ABB RobotStudio station: Proy_ROBG.rspag

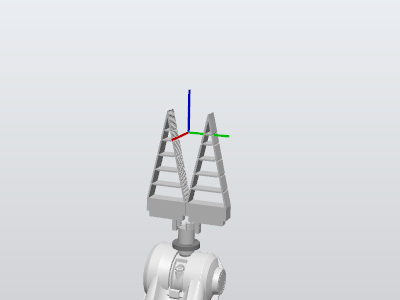
--- station ---
Station Project1 (saved by RobotStudio 23.3.10550.0)
Controller IRB140_6_81
  mechanical unit ROB_1: IRB140_6_81_C_03, 6 joints, base frame (0, 0, 0) mm
Layout (positions relative to the parent item):
  - IRB140_6_81_C_03 [mechanism, from %ABB.RobotStudio.Models.IRB140%\IRB140_6_81_C_G_03.rslib] at (0, 0, 0) mm; joint values [0, 0, -2.1624, 0, 0.5236, 0] (rad or m)
  - BandaViejita [part] at (100, -700, 100) mm, rotated rx 90 ry 0 rz -90 deg, size 200 x 230 x 1970 mm
  - Armario [part] at (750, -300, 50) mm, rotated rx 90 ry 0 rz 90 deg, size 600 x 1160 x 250 mm
  - SC_obj [smart component]
      signals: DI coger, DI soltar, AI pose
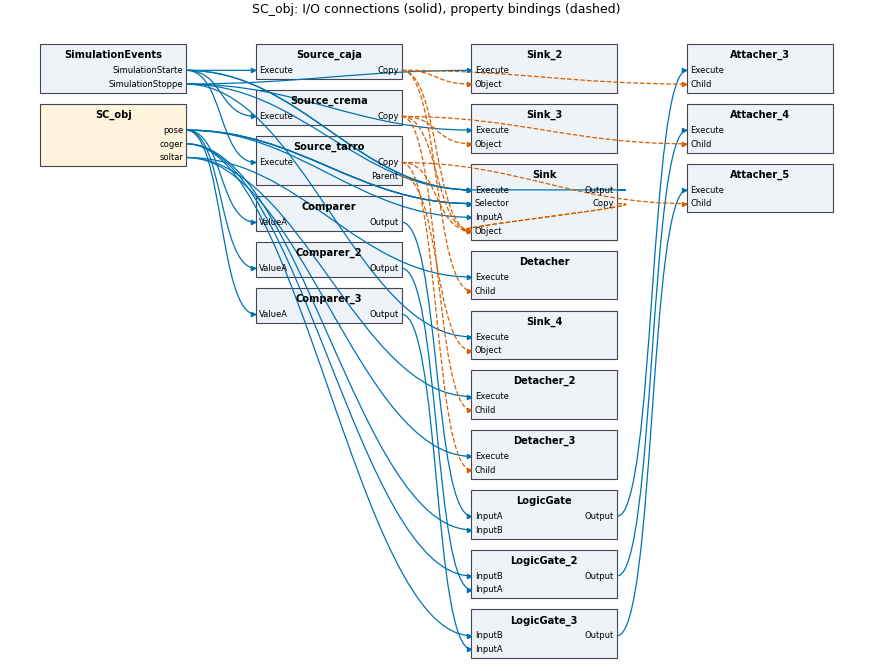
      connections:
        SimulationEvents.SimulationStarted -> Source_caja.Execute
        SimulationEvents.SimulationStopped -> Sink.Execute
        SimulationEvents.SimulationStarted -> Source_2.Execute
        SimulationEvents.SimulationStarted -> Source_3.Execute
        SC_obj.pose -> LogicMux.Selector
        SC_obj.pose -> LogicMux.InputA
        SC_obj.pose -> LogicMux_2.Selector
        LogicMux_3.Output -> Sink.Execute
        SC_obj.pose -> LogicMux_3.Selector
        SC_obj.pose -> Comparer.ValueA
        Comparer.Output -> LogicGate.InputA
        SC_obj.coger -> LogicGate.InputB
        LogicGate.Output -> Attacher_3.Execute
        SimulationEvents.SimulationStarted -> Source_crema.Execute
        SimulationEvents.SimulationStarted -> Source_tarro.Execute
        SC_obj.soltar -> Detacher.Execute
        SC_obj.soltar -> Detacher_2.Execute
        SC_obj.soltar -> Detacher_3.Execute
        SC_obj.coger -> LogicGate_2.InputB
        SC_obj.coger -> LogicGate_3.InputB
        Comparer_2.Output -> LogicGate_2.InputA
        Comparer_3.Output -> LogicGate_3.InputA
        SC_obj.pose -> Comparer_2.ValueA
        SC_obj.pose -> Comparer_3.ValueA
        LogicGate_2.Output -> Attacher_4.Execute
        LogicGate_3.Output -> Attacher_5.Execute
        SimulationEvents.SimulationStopped -> Sink_2.Execute
        SimulationEvents.SimulationStopped -> Sink_4.Execute
        SimulationEvents.SimulationStopped -> Sink_3.Execute
        Source_caja.Copy => Sink.Object
        Source_2.Copy => Sink.Object
        Source_3.Copy => Sink.Object
        Source_caja.Copy => Detacher.Child
        Source_caja.Copy => Attacher_3.Child
        Source_tarro.Copy => Sink.Object
        Source_crema.Copy => Sink.Object
        Source_crema.Copy => Attacher_4.Child
        Source_tarro.Copy => Attacher_5.Child
        Source_crema.Copy => Detacher_2.Child
        Source_tarro.Copy => Detacher_3.Child
        Source_caja.Copy => Sink_2.Object
        Source_crema.Copy => Sink_3.Object
        Source_tarro.Parent => Sink_4.Object
    - Caja [part] at (768.01, 178.37, 524.54) mm, rotated rx 0 ry 0 rz -87.57 deg, size 30 x 75 x 130 mm
    - Source_caja [smart component, from Components\Source.rslib]
        properties: Source=Caja; Copy=(none); Parent=(none); Position=[0.77 0.14 0.524544]; Orientation=[0 0 -1.5707963267949]; Transient=true; PhysicsBehavior=3
    - SimulationEvents [smart component, from Components\SimulationEvents.rslib]
    - planB [mechanism] at (-146.33, 0, 1092.27) mm, rotated rx 0 ry -3.89 rz 0 deg
        TCP planB at (0, 200, 0) mm, rotated rx -90 ry -30 rz 0 deg
        links: PlanB
    - Attacher_3 [smart component, from Components\Attacher.rslib]
        properties: Parent=planB; Flange=0; Child=(none); Mount=false; Offset=[0 0 0]; Orientation=[0 0 0]
    - Detacher [smart component, from Components\Detacher.rslib]
        properties: Child=(none); KeepPosition=false
    - Comparer [smart component, from Components\Comparer.rslib]
        properties: ValueA=3; Operator===; ValueB=1
    - LogicGate [smart component, from Components\LogicGate.rslib]
        properties: Operator=AND; Delay=0
    - LogicGate_2 [smart component, from Components\LogicGate.rslib]
        properties: Operator=AND; Delay=0
    - Crema [part] at (799.98, 0, 524.64) mm, rotated rx 90 ry 0 rz 90.03 deg, size 55 x 140 x 33 mm
    - Tarro [part] at (799.07, -184.56, 524.28) mm, rotated rx 90 ry 0 rz -4.09 deg, size 47 x 95 x 47 mm
    - Source_tarro [smart component, from Components\Source.rslib]
        properties: Source=Tarro; Copy=(none); Parent=(none); Position=[0.77 -0.14 0.524544]; Orientation=[1.5707963267949 0 -1.5707963267949]; Transient=true; PhysicsBehavior=3
    - Source_crema [smart component, from Components\Source.rslib]
        properties: Source=Crema; Copy=(none); Parent=(none); Position=[0.77 -0.14 0.25]; Orientation=[1.5707963267949 0 -1.5707963267949]; Transient=true; PhysicsBehavior=3
    - LogicGate_3 [smart component, from Components\LogicGate.rslib]
        properties: Operator=AND; Delay=0
    - Detacher_2 [smart component, from Components\Detacher.rslib]
        properties: Child=(none); KeepPosition=false
    - Detacher_3 [smart component, from Components\Detacher.rslib]
        properties: Child=(none); KeepPosition=false
    - Attacher_4 [smart component, from Components\Attacher.rslib]
        properties: Parent=planB; Flange=0; Child=(none); Mount=false; Offset=[0 0 0]; Orientation=[0 0 0]
    - Attacher_5 [smart component, from Components\Attacher.rslib]
        properties: Parent=planB; Flange=0; Child=(none); Mount=false; Offset=[0 0 0]; Orientation=[0 0 0]
    - Comparer_2 [smart component, from Components\Comparer.rslib]
        properties: ValueA=3; Operator===; ValueB=6
    - Comparer_3 [smart component, from Components\Comparer.rslib]
        properties: ValueA=3; Operator===; ValueB=3
    - Sink_2 [smart component, from Components\Sink.rslib]
        properties: Object=(none)
    - Sink_3 [smart component, from Components\Sink.rslib]
        properties: Object=(none)
    - Sink_4 [smart component, from Components\Sink.rslib]
        properties: Object=(none)
Attachment: planB is attached to IRB140_6_81_C_03 / Link6
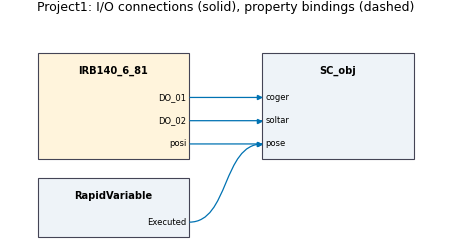
Station logic (signal -> signal, property => property):
  IRB140_6_81.DO_01 -> SC_obj.coger
  IRB140_6_81.DO_02 -> SC_obj.soltar
  RapidVariable.Executed -> SC_obj.pose
  IRB140_6_81.posi -> SC_obj.pose

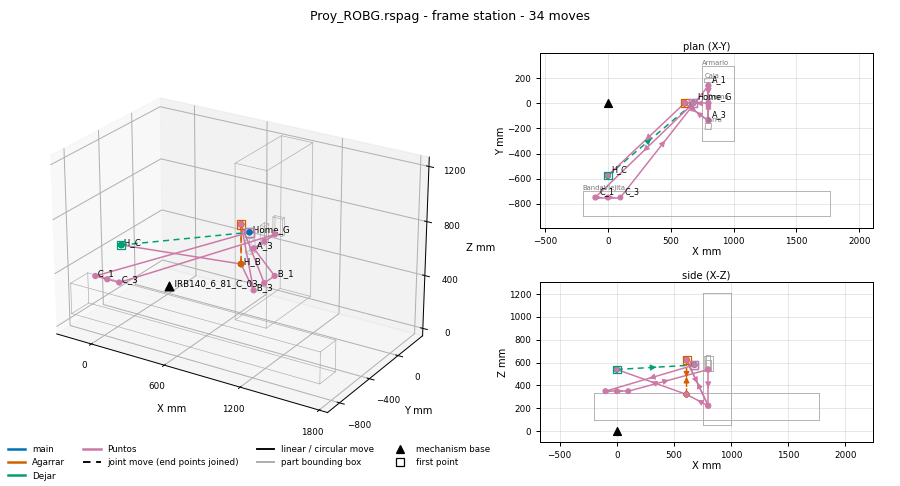
[picture p0: tool path of Proy_ROBG.rspag in frame station, 34 of 40 moves have a stored position in this frame; points joined in program order, loops and branches not executed]
--- Controller Data/IRB140_6_81/RAPID/TASK1/PROGMOD/CalibData.mod ---
MODULE CalibData
ENDMODULE

--- Controller Data/IRB140_6_81/RAPID/TASK1/PROGMOD/Module1.mod ---
MODULE Module1
    CONST robtarget C_1:=[[100,150,20],[0.5,0.5,0.5,-0.5],[-2,-1,1,1],[9E+09,9E+09,9E+09,9E+09,9E+09,9E+09]];
    CONST robtarget C_2:=[[200,150,20],[0.5,0.5,0.5,-0.5],[-1,-1,1,1],[9E+09,9E+09,9E+09,9E+09,9E+09,9E+09]];
    CONST robtarget C_3:=[[300,150,20],[0.5,0.5,0.5,-0.5],[-1,0,0,1],[9E+09,9E+09,9E+09,9E+09,9E+09,9E+09]];
    VAR signaldi Pos_dejar;
    TASK PERS wobjdata W_Banda:=[FALSE,TRUE,"",[[0,0,100],[1,0,0,0]],[[-200,-900,230],[1,0,0,0]]];
    CONST robtarget Home_G:=[[679.496732003,0,579.5],[0.5,0,0.866025404,0],[0,0,0,0],[9E+09,9E+09,9E+09,9E+09,9E+09,9E+09]];
    CONST robtarget A_1:=[[140,50,20],[0.5,-0.5,0.5,0.5],[0,0,-2,1],[9E+09,9E+09,9E+09,9E+09,9E+09,9E+09]];
    CONST robtarget A_2:=[[280,50,20],[0.5,-0.5,0.5,0.5],[0,0,-1,1],[9E+09,9E+09,9E+09,9E+09,9E+09,9E+09]];
    CONST robtarget A_3:=[[420,50,20],[0.5,-0.5,0.5,0.5],[-1,-1,-1,1],[9E+09,9E+09,9E+09,9E+09,9E+09,9E+09]];
    CONST robtarget B_1:=[[140,50,-297.5],[0.5,-0.5,0.5,0.5],[0,0,-2,1],[9E+09,9E+09,9E+09,9E+09,9E+09,9E+09]];
    CONST robtarget B_2:=[[280,50,-297.5],[0.5,-0.5,0.5,0.5],[0,0,-1,1],[9E+09,9E+09,9E+09,9E+09,9E+09,9E+09]];
    CONST robtarget B_3:=[[420,50,-297.5],[0.5,-0.5,0.5,0.5],[-1,-1,-1,1],[9E+09,9E+09,9E+09,9E+09,9E+09,9E+09]];
    TASK PERS wobjdata W_Armario:=[FALSE,TRUE,"",[[750,280,520],[0.707107,0,0,-0.707107]],[[0,0,0],[1,0,0,0]]];
    CONST robtarget H_A:=[[280,-139.508914925,103.770212837],[0.5,-0.5,0.5,0.5],[0,0,-1,1],[9E+09,9E+09,9E+09,9E+09,9E+09,9E+09]];
    CONST robtarget H_B:=[[280,-139.933171273,-197.954698627],[0.5,-0.5,0.5,0.5],[0,0,-1,1],[9E+09,9E+09,9E+09,9E+09,9E+09,9E+09]];
    CONST robtarget H_C:=[[199.999965031,324.731782319,210.32453317],[0.5,0.5,0.5,-0.5],[-2,-1,1,1],[9E+09,9E+09,9E+09,9E+09,9E+09,9E+09]];
    PERS num op_agarrar:=3;
    PERS num op_dejar:=3;
    PERS bool flag_A1:=FALSE;
    PERS bool flag_A2:=FALSE;
    PERS bool flag_A3:=FALSE;
    PERS bool flag_B1:=FALSE;
    PERS bool flag_B2:=FALSE;
    PERS bool flag_B3:=FALSE;
    PERS bool flag_C1:=FALSE;
    PERS bool flag_C2:=FALSE;
    PERS bool flag_C3:=FALSE;
    PERS tooldata planB:=[TRUE,[[0,0,200],[1,0,0,0]],[1,[0,0,1],[1,0,0,0],0,0,0]];
    LOCAL PERS tooldata Servo:=[TRUE,[[0,0,114.2],[1,0,0,0]],[0.215,[8.7,12.3,49.2],[1,0,0,0],0.00021,0.00024,0.00009]];


    !***********************************************************
    !
    ! M?dulo:  Module1
    !
    ! Descripción:
    !   <Introduzca la descripción aquí>
    !
    ! Autor: gio
    !
    ! Versión: 1.0
    !
    !***********************************************************


    !***********************************************************
    !
    ! Procedimiento Main
    !
    !   Este es el punto de entrada de su programa
    !
    !***********************************************************
    PROC main()
        !Add your code here
        inicio:
        WaitDO DO_03,1;
        MoveJ Home_G,v300,z5,planB\WObj:=wobj0;
        setAO posi, op_agarrar;
        Agarrar op_agarrar,[0,-100,0],TRUE;
        Dejar op_dejar,[0,0,100],FALSE;
        GOTO inicio;
    ENDPROC
PROC Agarrar(num option, pos offset, bool d)
    ! Realizar acciones basadas en la opción seleccionada
    TEST option
        CASE 1:
            ! Realizar acción para la opción 1
            flag_A1:=True;
            MoveJ H_A,v500,z5,planB\WObj:=W_Armario;
            Move_offset A_1, offset, FALSE, d;
            MoveL H_A,v500,z5,planB\WObj:=W_Armario;
        CASE 2:
            ! Realizar acción para la opción 2
            flag_A2:=True;
            MoveJ H_A,v500,z5,planB\WObj:=W_Armario;
            Move_offset A_2, offset, FALSE, d;
            MoveJ H_A,v500,z5,planB\WObj:=W_Armario;
        CASE 3:
            ! Realizar acción para la opción 3
            flag_A3:=True;
            MoveJ H_A,v500,z5,planB\WObj:=W_Armario;
            Move_offset A_3, offset, FALSE, d;
            MoveJ H_A,v500,z5,planB\WObj:=W_Armario;
        CASE 4:
            ! Realizar acción para la opción 1
            flag_B1:=True;
            MoveJ H_B,v500,z5,planB\WObj:=W_Armario;
            Move_offset B_1, offset, FALSE, d;
            MoveJ H_B,v500,z5,planB\WObj:=W_Armario;
        CASE 5:
            ! Realizar acción para la opción 2
            flag_B2:=True;
            MoveJ H_B,v500,z5,planB\WObj:=W_Armario;
            Move_offset B_2, offset, FALSE, d;
            MoveJ H_B,v500,z5,planB\WObj:=W_Armario;
        CASE 6:
            ! Realizar acción para la opción 3
            flag_B3:=True;
            MoveJ H_B,v500,z5,planB\WObj:=W_Armario;
            Move_offset B_3, offset, FALSE, d;
            MoveJ H_B,v500,z5,planB\WObj:=W_Armario;
        DEFAULT:
            ! Manejar caso donde la opción no es válida
    ENDTEST
        MoveJ H_A,v500,z5,planB\WObj:=W_Armario;
        apagarFlag;
   ENDPROC
PROC Dejar(num option, pos offset,bool d)
    ! Realizar acciones basadas en la opción seleccionada
    TEST option
        CASE 1:
            ! Realizar acción para la opción 1
            flag_C1:=True;
            MoveJ H_C,v500,z5,planB\WObj:=W_Banda;
            Move_offset C_1, offset, TRUE, d;
            MoveJ H_C,v500,z5,planB\WObj:=W_Banda;
        CASE 2:
            ! Realizar acción para la opción 2
            flag_C2:=True;
            MoveJ H_C,v500,z5,planB\WObj:=W_Banda;
            Move_offset C_2, offset, TRUE, d;
            MoveJ H_C,v500,z5,planB\WObj:=W_Banda;
        CASE 3:
            ! Realizar acción para la opción 3
            flag_C3:=True;
            MoveJ H_C,v500,z5,planB\WObj:=W_Banda;
            Move_offset C_3, offset, TRUE, d;
            MoveJ H_C,v500,z5,planB\WObj:=W_Banda;
        DEFAULT:
            ! Manejar caso donde la opción no es válida
    ENDTEST
        MoveJ Home_G,v500,z5,planB\WObj:=wobj0;
        apagarFlag;
   ENDPROC



PROC Move_offset(robtarget target, pos offset,bool W, bool d)
    ! Moverse a 100 mm por encima del punto
    IF W THEN
        MoveL Offs (target, offset.x, offset.y, offset.z), v500, z5, planB\WObj:=W_Banda;
        ! Bajar linealmente al punto
        MoveL target, v50, z5, planB\WObj:=W_banda;
    ELSE
        MoveL Offs (target, offset.x, offset.y, offset.z), v500, z5, planB\WObj:=W_Armario;
        ! Bajar linealmente al punto
        MoveL target, v50, z5, planB\WObj:=W_Armario;
    ENDIF
    WaitTime 1;
    ! Activar o Desactivar la entrada digital número
    IF d THEN
        SetDO DO_01, 1;
        WaitTime 1;
        SetDO DO_01, 0;
    ELSE
        SetDO DO_02, 1;
        WaitTime 1;
        SetDO DO_02, 0;
    ENDIF
    WaitTime 5;
    ! Volver a subir
    IF W THEN
        MoveL Offs (target, offset.x, offset.y, offset.z), v50, z5, planB\WObj:=W_Banda;
    ELSE
        MoveL Offs (target, offset.x, offset.y, offset.z), v50, z5, planB\WObj:=W_Armario;
    ENDIF
ENDPROC
PROC apagarFlag()
    flag_A1:=False;
    flag_A2:=False;
    flag_A3:=False;
    flag_B1:=False;
    flag_B2:=False;
    flag_B3:=False;
    flag_C1:=False;
    flag_C2:=False;
    flag_C3:=False;
ENDPROC


    LOCAL PROC Puntos()
        MoveL Home_G,v500,z5,planB\WObj:=wobj0;
        MoveL C_1,v500,z5,planB\WObj:=W_Banda;
        MoveL C_2,v500,z5,planB\WObj:=W_Banda;
        MoveL C_3,v500,z5,planB\WObj:=W_Banda;
        MoveL A_1,v500,z5,planB\WObj:=W_Armario;
        MoveL A_2,v500,z5,planB\WObj:=W_Armario;
        MoveL A_3,v500,z5,planB\WObj:=W_Armario;
        MoveL B_1,v500,z5,planB\WObj:=W_Armario;
        MoveL B_2,v500,z5,planB\WObj:=W_Armario;
        MoveL H_A,v500,z5,planB\WObj:=W_Armario;
        MoveL B_3,v500,z5,planB\WObj:=W_Armario;
        MoveL H_B,v500,z5,planB\WObj:=W_Armario;
        MoveL H_C,v500,z5,planB\WObj:=W_Banda;
    ENDPROC

ENDMODULE

--- Controller Data/IRB140_6_81/SYSPAR/EIO.cfg ---
EIO:CFG_1.0:6:1::
#
EIO_SIGNAL:

      -Name "DO_02" -SignalType "DO" -Access "All"

      -Name "DO_01" -SignalType "DO" -Access "All"

      -Name "DO_03" -SignalType "DO" -Access "All"

      -Name "posi" -SignalType "AO" -Access "All" -EncType "UNSIGNED"
